// TIA Portal V16 export
// export: Created 2023-03-29T11:04:47.374941Z, ExportSetting WithDefaults, DisplayName Totally Integrated Automation Portal, DisplayVersion V16 Update 6, DisplayName TIA Portal Version Control Interface, DisplayVersion V16 Update 2, DisplayName TIA Portal Openness, DisplayVersion V16 Update 6, DisplayName STEP 7 Professional, DisplayVersion V16 Update 6, DisplayName STEP 7 Safety, DisplayVersion V16, DisplayName WinCC Advanced, DisplayVersion V16 Update 6
DATA_BLOCK "Czasy pracy DM"   // DB30
{ S7_Optimized_Access := 'FALSE' }
VERSION : 0.1
// stored: AutoNumber false, DBAccessibleFromOPCUA true, IsOnlyStoredInLoadMemory false, IsWriteProtectedInAS false
   VAR
      Sek_P1 : Int := 1;   // Licznik sekund
      Sek_P2 : Int := 2;   // Licznik sekund
      Sek_P3 : Int := 3;   // Licznik sekund
      Sek_P4 : Int := 3;
      Edge_P1 : Bool;   // Pamięć zbocza
      Edge_P2 : Bool;   // Pamięć zbocza
      Edge_P3 : Bool;   // Pamięć zbocza
      Edge_P4 : Bool := false;
      Sek_a : Int;   // Licznik sekund
      Sek_b : Int;   // Licznik sekund
      Edge_a : Bool;   // Pamięć zbocza
      Edge_b : Bool;   // Pamięć zbocza
      Sum_sek_hur_P1 : Real;   // Licznik sumator godzin i sekund na potrzeby wyznaczania dumchawy do pracy
      Sum_sek_hur_P2 : Real := 0.0;   // Licznik sumator godzin i sekund na potrzeby wyznaczania dumchawy do pracy
      Sum_sek_hur_P3 : Real := 0.0;   // Licznik sumator godzin i sekund na potrzeby wyznaczania dumchawy do pracy
      Sum_sek_hur_P4 : Real := 0.0;
   END_VAR
BEGIN
END_DATA_BLOCK
